SUBAPPLICATION SlurryTanker (* Subapplication Type *)
  (* Standard: 61499-2 *)
  (* Version 1.0, 2023-02-11, franz *)
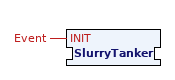
  EVENT_INPUT
    INIT;
  END_EVENT
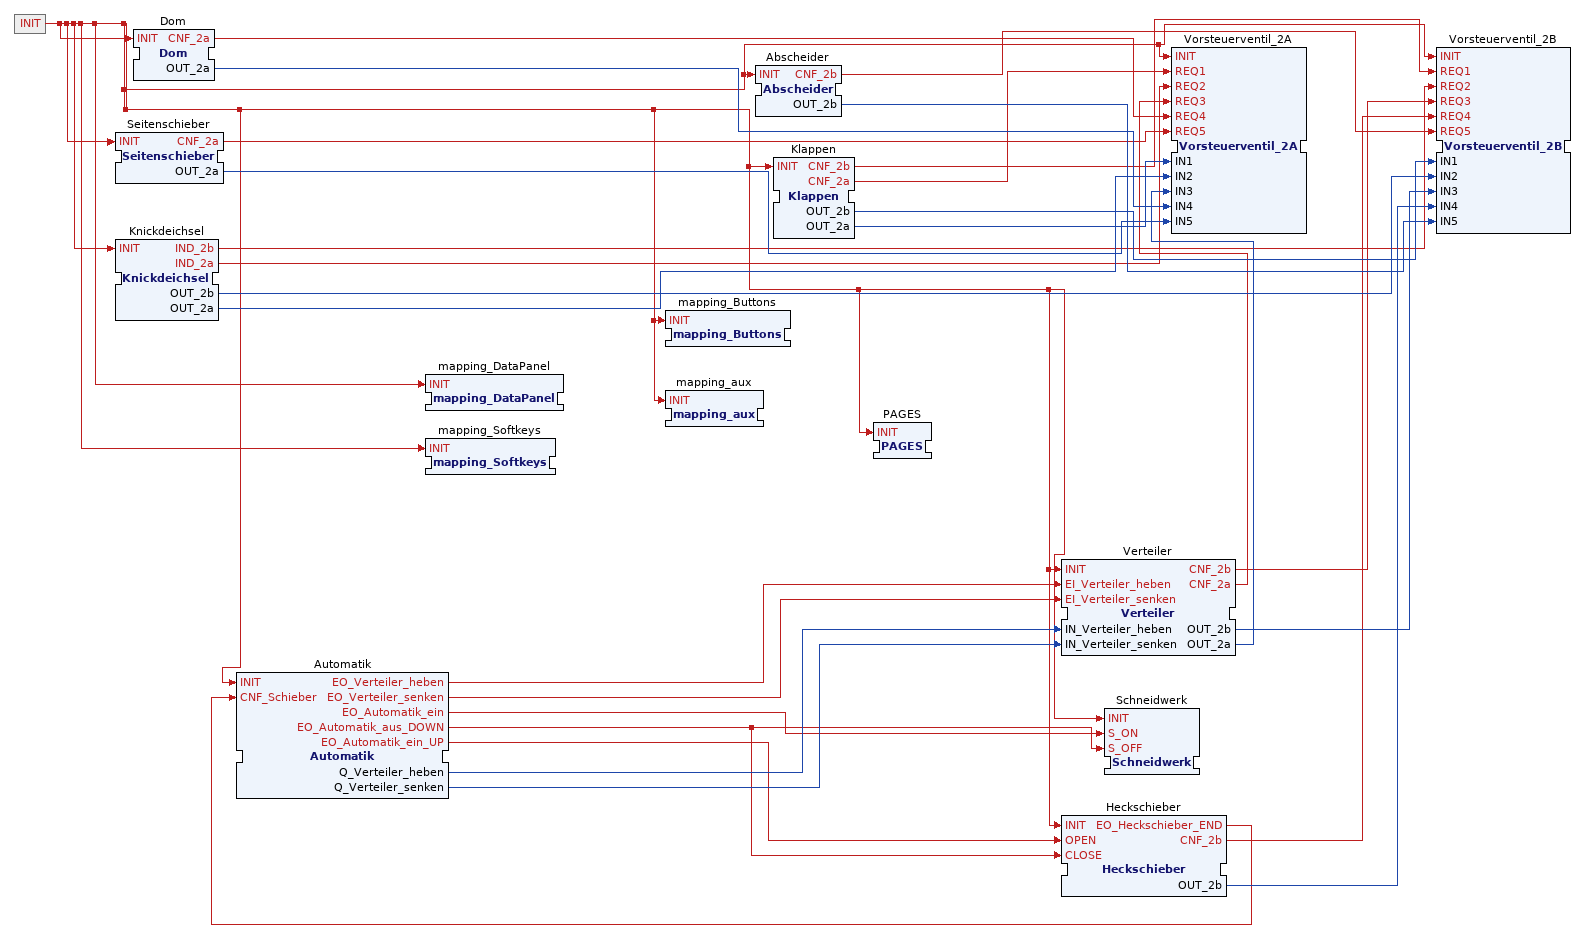
  (* Group func: *)
  (* Group Vorsteuerventile: Vorsteuerventile *)
  (* Group Vorgewendeautomatik: Vorgewendeautomatik *)
  SUBAPPS
    Vorsteuerventil_2A : Vorsteuerventil_2A; {SET_ATTRIBUTE(GroupName, Vorsteuerventile)}
    Vorsteuerventil_2B : Vorsteuerventil_2B; {SET_ATTRIBUTE(GroupName, Vorsteuerventile)}
    Dom : Dom; {SET_ATTRIBUTE(GroupName, func)}
    Seitenschieber : Seitenschieber; {SET_ATTRIBUTE(GroupName, func)}
    Knickdeichsel : Knickdeichsel; {SET_ATTRIBUTE(GroupName, func)}
    mapping_Softkeys : mapping_Softkeys; {SET_ATTRIBUTE(GroupName, func)}
    mapping_DataPanel : mapping_DataPanel; {SET_ATTRIBUTE(GroupName, func)}
    mapping_aux : mapping_aux; {SET_ATTRIBUTE(GroupName, func)}
    Automatik : Automatik; {SET_ATTRIBUTE(GroupName, Vorgewendeautomatik)}
    Verteiler : Verteiler; {SET_ATTRIBUTE(GroupName, Vorgewendeautomatik)}
    Schneidwerk : Schneidwerk; {SET_ATTRIBUTE(GroupName, Vorgewendeautomatik)}
    Heckschieber : Heckschieber; {SET_ATTRIBUTE(GroupName, Vorgewendeautomatik)}
    Abscheider : Abscheider; {SET_ATTRIBUTE(GroupName, func)}
    Klappen : Klappen; {SET_ATTRIBUTE(GroupName, func)}
    PAGES : PAGES; {SET_ATTRIBUTE(GroupName, func)}
    mapping_Buttons : mapping_Buttons; {SET_ATTRIBUTE(GroupName, func)}
  END_SUBAPPS
  EVENT_CONNECTIONS
    INIT TO Dom.INIT;
    INIT TO Seitenschieber.INIT;
    INIT TO Knickdeichsel.INIT;
    INIT TO mapping_Softkeys.INIT;
    INIT TO mapping_aux.INIT;
    INIT TO mapping_DataPanel.INIT;
    INIT TO Abscheider.INIT;
    INIT TO Klappen.INIT;
    INIT TO Vorsteuerventil_2A.INIT;
    INIT TO Vorsteuerventil_2B.INIT;
    INIT TO Verteiler.INIT;
    INIT TO Automatik.INIT;
    INIT TO Heckschieber.INIT;
    INIT TO Schneidwerk.INIT;
    Automatik.EO_Verteiler_heben TO Verteiler.EI_Verteiler_heben;
    Automatik.EO_Verteiler_senken TO Verteiler.EI_Verteiler_senken;
    Automatik.EO_Automatik_ein TO Schneidwerk.S_ON;
    Automatik.EO_Automatik_aus_DOWN TO Schneidwerk.S_OFF;
    Automatik.EO_Automatik_ein_UP TO Heckschieber.OPEN;
    Automatik.EO_Automatik_aus_DOWN TO Heckschieber.CLOSE;
    Heckschieber.EO_Heckschieber_END TO Automatik.CNF_Schieber;
    Klappen.CNF_2b TO Vorsteuerventil_2B.REQ1;
    Klappen.CNF_2a TO Vorsteuerventil_2A.REQ1;
    Knickdeichsel.IND_2b TO Vorsteuerventil_2B.REQ2;
    Knickdeichsel.IND_2a TO Vorsteuerventil_2A.REQ2;
    Verteiler.CNF_2b TO Vorsteuerventil_2B.REQ3;
    Verteiler.CNF_2a TO Vorsteuerventil_2A.REQ3;
    Heckschieber.CNF_2b TO Vorsteuerventil_2B.REQ4;
    Dom.CNF_2a TO Vorsteuerventil_2A.REQ4;
    Seitenschieber.CNF_2a TO Vorsteuerventil_2A.REQ5;
    Abscheider.CNF_2b TO Vorsteuerventil_2B.REQ5;
    INIT TO PAGES.INIT;
    INIT TO mapping_Buttons.INIT;
  END_CONNECTIONS
  DATA_CONNECTIONS
    Automatik.Q_Verteiler_heben TO Verteiler.IN_Verteiler_heben;
    Automatik.Q_Verteiler_senken TO Verteiler.IN_Verteiler_senken;
    Klappen.OUT_2b TO Vorsteuerventil_2B.IN1;
    Klappen.OUT_2a TO Vorsteuerventil_2A.IN1;
    Knickdeichsel.OUT_2b TO Vorsteuerventil_2B.IN2;
    Knickdeichsel.OUT_2a TO Vorsteuerventil_2A.IN2;
    Verteiler.OUT_2b TO Vorsteuerventil_2B.IN3;
    Verteiler.OUT_2a TO Vorsteuerventil_2A.IN3;
    Heckschieber.OUT_2b TO Vorsteuerventil_2B.IN4;
    Dom.OUT_2a TO Vorsteuerventil_2A.IN4;
    Seitenschieber.OUT_2a TO Vorsteuerventil_2A.IN5;
    Abscheider.OUT_2b TO Vorsteuerventil_2B.IN5;
  END_CONNECTIONS
END_SUBAPPLICATION
